Yaskawa INFORM job: pos_z_1.JBI

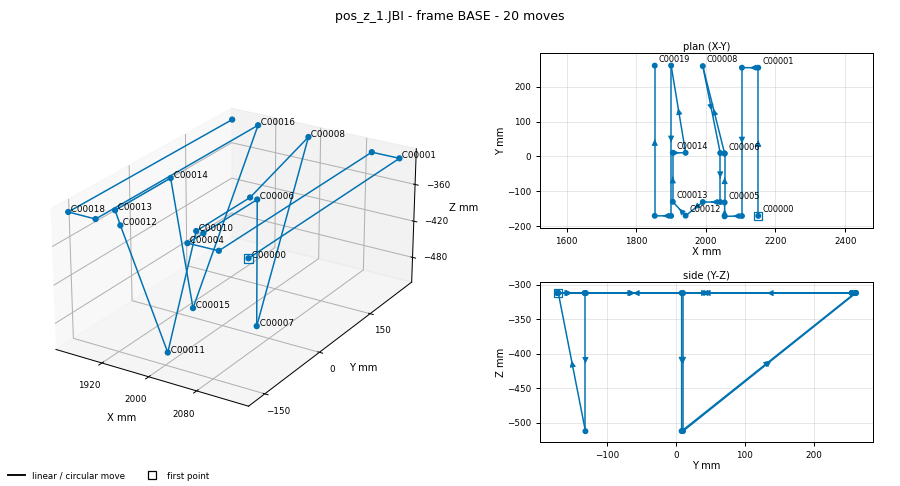
[picture p0: tool path of pos_z_1.JBI in frame BASE, 20 of 22 moves have a stored position in this frame; points joined in program order, loops and branches not executed]
/JOB
//NAME pos_z_1
//POS
///NPOS 20,0,20,0,0,0
///TOOL 0
///POSTYPE BASE
///RECTAN
///RCONF 0,0,0,0,0,0,0,0,0,0,0,0,0,0,0,0,0,0,0,0,0,0,0,0
C00000=2150.499142,-170.718890,-311.836795,-175.000000,-5.000000,-5.000000
C00001=2150.499142,254.705110,-311.836795,-175.000000,-5.000000,-5.000000
C00002=2103.679400,254.799372,-311.838353,-175.000000,5.000000,5.000000
C00003=2103.679400,-171.056628,-311.838353,-175.000000,5.000000,5.000000
C00004=2053.922199,-172.133646,-311.914010,-175.000000,5.000000,5.000000
C00005=2054.042199,-132.310646,-311.914225,-175.000000,5.000000,5.000000
C00006=2054.042199,8.405354,-311.914225,-175.000000,5.000000,5.000000
C00007=2053.922199,8.405654,-511.914010,-175.000000,5.000000,5.000000
C00008=1991.241004,259.354715,-312.077632,-175.000000,-5.000000,-5.000000
C00009=2041.361004,9.755715,-312.077848,-175.000000,-5.000000,-5.000000
C00010=2041.361004,-130.960285,-312.077848,-175.000000,-5.000000,-5.000000
C00011=1991.241004,-130.960285,-512.077632,-175.000000,-5.000000,-5.000000
C00012=1941.911808,-170.199961,-312.005490,-175.000000,-5.000000,-5.000000
C00013=1905.131808,-130.324961,-312.005706,-175.000000,-5.000000,-5.000000
C00014=1905.131808,10.391039,-312.005706,-175.000000,-5.000000,-5.000000
C00015=1941.911808,10.391339,-512.005490,-175.000000,-5.000000,-5.000000
C00016=1900.324174,260.964496,-311.813349,-175.000000,-5.000000,-5.000000
C00017=1900.324174,-170.738504,-311.813349,-175.000000,-5.000000,-5.000000
C00018=1853.284352,-170.551172,-311.825600,-175.000000,5.000000,5.000000
C00019=1853.284352,260.724828,-311.825600,-175.000000,5.000000,5.000000
///POSTYPE PULSE
///PULSE
EX000=0
///POSTYPE PULSE
///PULSE
EC00000=0
EC00001=0
EC00002=0
EC00003=0
EC00004=0
EC00005=0
EC00006=0
EC00007=0
EC00008=0
EC00009=0
EC00010=0
EC00011=0
EC00012=0
EC00013=0
EC00014=0
EC00015=0
EC00016=0
EC00017=0
EC00018=0
EC00019=0
//INST
///DATE 2023/06/26 11:09
///ATTR SC,RW,RJ
////FRAME BASE
///GROUP1 RB1,ST1
NOP
MOVJ P009 EX000 VJ=15.00
MOVJ C00000 EC00000 VJ=15.0
CALL JOB:SPYON
MOVL C00001 EC00001 V=150.0
MOVL C00002 EC00002 V=150.0
MOVL C00003 EC00003 V=150.0
MOVL C00004 EC00004 V=150.0
CALL JOB:SPYOF
MOVL C00005 EC00005 V=150.0
MOVL C00006 EC00006 V=150.0
MOVL C00007 EC00007 V=150.0
CALL JOB:SPYON
MOVL C00008 EC00008 V=150.0
CALL JOB:SPYOF
MOVL C00009 EC00009 V=150.0
MOVL C00010 EC00010 V=150.0
MOVL C00011 EC00011 V=150.0
CALL JOB:SPYON
MOVL C00012 EC00012 V=150.0
CALL JOB:SPYOF
MOVL C00013 EC00013 V=150.0
MOVL C00014 EC00014 V=150.0
MOVL C00015 EC00015 V=150.0
CALL JOB:SPYON
MOVL C00016 EC00016 V=150.0
MOVL C00017 EC00017 V=150.0
MOVL C00018 EC00018 V=150.0
MOVL C00019 EC00019 V=150.0
CALL JOB:SPYOF
MOVJ P009 VJ=15.00
END
